VAR_GLOBAL
	
SR110_Vert_servo_ctrl:Servo_Control;
	SR110_Vert_servo_status:stManualModeAxis;
	OP110_HMI_Reset:						    BOOL;
END_VAR

(* stored: Version 1.1.0.1, ProductVersion 3.1.4024.11
   GVL OP110_HMI_GVL: Id {577cebaf-abb8-4306-a2bf-ae3b7d67c9fd} *)
